PROGRAM MAIN
VAR
    cola:FB_piec; 
    czasoOpuzniacz:TON;
END_VAR

czasoOpuzniacz(IN:=TRUE,PT:=T#10MS);
IF  czasoOpuzniacz.Q=TRUE AND DVL.stanprzycisku=TRUE THEN
    cola();
    czasoOpuzniacz(IN:=FALSE);
END_IF

END_PROGRAM

(* stored: Version 1.1.0.1, ProductVersion 3.1.4024.4
   POU MAIN: Id {18596b13-74dd-4adc-9fd9-0da5bf571f0e}, SpecialFunc None *)
